TYPE DUT_Test :
STRUCT
	value: BOOL;
	abc: DUT_Test_1;
END_STRUCT
END_TYPE

(* stored: Version 1.1.0.1, ProductVersion 3.1.4024.11
   DUT DUT_Test: Id {de0ddf2a-28fa-495d-a74c-09d6bc088d93} *)
